   IF "Modbus_Buffer".Time_Venting <> 0 AND "Modbus_Buffer".Time_Venting <> "Torche_DB".Signal_Torche.Time_vent_g THEN
           "Torche_DB".Signal_Torche.Time_vent_g := "Modbus_Buffer".Time_Venting;
       END_IF;
       IF "Modbus_Buffer".Time_firing <> 0 AND "Modbus_Buffer".Time_firing <> "Torche_DB".Signal_Torche.Time_firing_g THEN
           "Torche_DB".Signal_Torche.Time_firing_g := "Modbus_Buffer".Time_firing;
       END_IF;
       IF "Modbus_Buffer".Time_spark_on <> 0 AND "Modbus_Buffer".Time_spark_on <> "Torche_DB".Signal_Torche.Time_spark_on_g THEN
           "Torche_DB".Signal_Torche.Time_spark_on_g := "Modbus_Buffer".Time_spark_on;
       END_IF;
       IF "Modbus_Buffer".Time_spark_off <> 0 AND "Modbus_Buffer".Time_spark_off <> "Torche_DB".Signal_Torche.Time_spark_off_g THEN
           "Torche_DB".Signal_Torche.Time_spark_off_g := "Modbus_Buffer".Time_spark_off;
       END_IF;
       IF "Modbus_Buffer".Time_stabil <> 0 AND "Modbus_Buffer".Time_stabil <> "Torche_DB".Signal_Torche.Time_stabiliz_g THEN
           "Torche_DB".Signal_Torche.Time_stabiliz_g := "Modbus_Buffer".Time_stabil;
       END_IF;
       IF "Modbus_Buffer".Time_after_alarm <> 0 AND "Modbus_Buffer".Time_after_alarm <> "Torche_DB".Signal_Torche.Time_after_alm_g  THEN
           "Torche_DB".Signal_Torche.Time_after_alm_g:= "Modbus_Buffer".Time_after_alarm;
       END_IF;
       IF "Modbus_Buffer".Time_after_stop <> 0 AND "Modbus_Buffer".Time_after_stop <> "Torche_DB".Signal_Torche.Time_stop_fire_g THEN
           "Torche_DB".Signal_Torche.Time_stop_fire_g := "Modbus_Buffer".Time_after_stop;
       END_IF;

       IF "Modbus_Buffer".Temp_Fire <> 0 AND "Modbus_Buffer".Temp_Fire <> "Temp_gorelka".Signal_AI.HH_Lim THEN
           "Temp_gorelka".Signal_AI.HH_Lim := "Modbus_Buffer".Temp_Fire;
       END_IF;
       IF "Modbus_Buffer".Temp_Fire <> 0 AND "Modbus_Buffer".Temp_Fire <> "temp_gorelka_2".Signal_AI.HH_Lim THEN
           "temp_gorelka_2".Signal_AI.HH_Lim := "Modbus_Buffer".Temp_Fire;
       END_IF;
       IF "Modbus_Buffer".Scal_max <> 0 AND "Modbus_Buffer".Scal_max <> "Temp_gorelka".Signal_AI.Scal_Max_Eu THEN
           "Temp_gorelka".Signal_AI.Scal_Max_Eu := "Modbus_Buffer".Scal_max;
       END_IF;
       IF "Modbus_Buffer".Scal_max <> 0 AND "Modbus_Buffer".Scal_max <> "temp_gorelka_2".Signal_AI.Scal_Max_Eu THEN
           "temp_gorelka_2".Signal_AI.Scal_Max_Eu := "Modbus_Buffer".Scal_max;
       END_IF;
       IF "Modbus_Buffer".Scal_min <> 0 AND "Modbus_Buffer".Scal_min <> "Temp_gorelka".Signal_AI.Scal_Min_Eu THEN
           "Temp_gorelka".Signal_AI.Scal_Min_Eu := "Modbus_Buffer".Scal_min;
       END_IF;
       IF "Modbus_Buffer".Scal_min <> 0 AND "Modbus_Buffer".Scal_min <> "temp_gorelka_2".Signal_AI.Scal_Min_Eu THEN
           "temp_gorelka_2".Signal_AI.Scal_Min_Eu := "Modbus_Buffer".Scal_min;
       END_IF;




   //********************ФОрмирование команды: запуск факела с верхнего уровня
   IF NOT "Modbus_Buffer".Start THEN
       "MB_Start" := false;
   ELSIF "Modbus_Buffer".Start THEN
       "MB_Start" := true;
       "Modbus_Buffer".Start := false;
   END_IF;

   IF NOT "Modbus_Buffer".Stop THEN
       "MB_Stop" := false;
   ELSIF "Modbus_Buffer".Stop THEN
       "MB_Stop" := true;
       "Modbus_Buffer".Stop := false;
   END_IF;

   IF NOT "Modbus_Buffer".Temp_curr_voltage THEN
       "Temp_gorelka".Signal_AI.VoltageInputType := false;
   ELSIF "Modbus_Buffer".Temp_curr_voltage THEN
       "Temp_gorelka".Signal_AI.VoltageInputType := true;
   END_IF;

   IF NOT "Modbus_Buffer".Temp_curr_voltage THEN
       "temp_gorelka_2".Signal_AI.VoltageInputType := false;
   ELSIF "Modbus_Buffer".Temp_curr_voltage THEN
       "temp_gorelka_2".Signal_AI.VoltageInputType := true;
   END_IF;
END_FUNCTION

// folder: PROFINET

FUNCTION "PUT" : Void   // FC9, SCL
{ S7_Optimized_Access := 'TRUE' }
VERSION : 0.1
BEGIN
   //"PN_XCHANGE_DB".AI1_Ch1 := "PT200".Signal_AI;
   //"PN_XCHANGE_DB".AI1_Ch2 := "TT200".Signal_AI;
   //"PN_XCHANGE_DB".AI1_Ch3 := "LT200_1".Signal_AI;
   //нужно дописать перемещение всех данных и заполнить PN_XCHANGE_DB
END_FUNCTION

FUNCTION "GET" : Void   // FC12, SCL
{ S7_Optimized_Access := 'TRUE' }
VERSION : 0.1
BEGIN
   //"PT200".Signal_AI := "PN_XCHANGE_DB".AI1_Ch1;
   // Заполнить до конца, разобраться когда вызывать эту функцию и функцию PUT
END_FUNCTION

FUNCTION "FC_SEND" : Void   // FC100, FBD
{ S7_Optimized_Access := 'TRUE' }
VERSION : 0.1
BEGIN

REGION Network 1
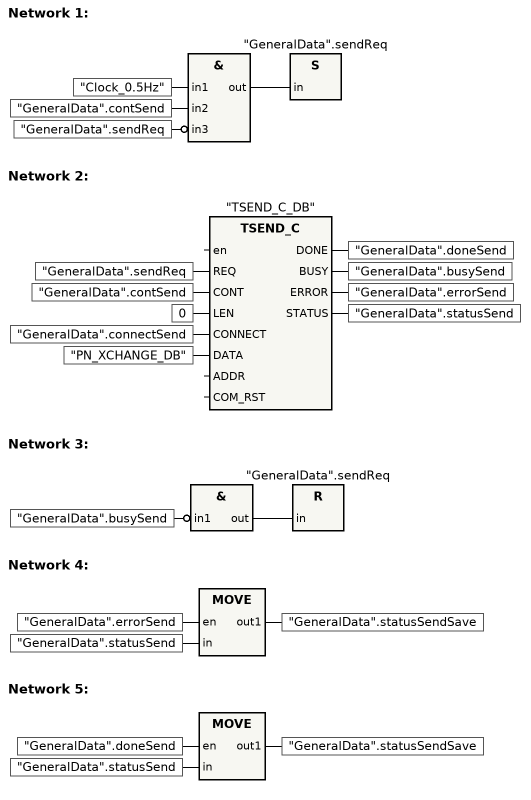
   IF "Clock_0.5Hz" AND "GeneralData".contSend AND NOT "GeneralData".sendReq THEN
       "GeneralData".sendReq := TRUE;
   END_IF;
END_REGION

REGION Network 2
   "TSEND_C_DB"(REQ := "GeneralData".sendReq,   // TSEND_C
                CONT := "GeneralData".contSend,
                LEN := 0,
                CONNECT := "GeneralData".connectSend,
                DATA := "PN_XCHANGE_DB",
                DONE => "GeneralData".doneSend,
                BUSY => "GeneralData".busySend,
                ERROR => "GeneralData".errorSend,
                STATUS => "GeneralData".statusSend);
END_REGION

REGION Network 3
   IF NOT "GeneralData".busySend THEN "GeneralData".sendReq := FALSE; END_IF;
END_REGION

REGION Network 4
   IF "GeneralData".errorSend THEN "GeneralData".statusSendSave := "GeneralData".statusSend; END_IF;
END_REGION

REGION Network 5
   IF "GeneralData".doneSend THEN "GeneralData".statusSendSave := "GeneralData".statusSend; END_IF;
END_REGION
END_FUNCTION

FUNCTION "FC_RECV" : Void   // FC200, FBD
{ S7_Optimized_Access := 'TRUE' }
VERSION : 0.1
BEGIN

REGION Network 1
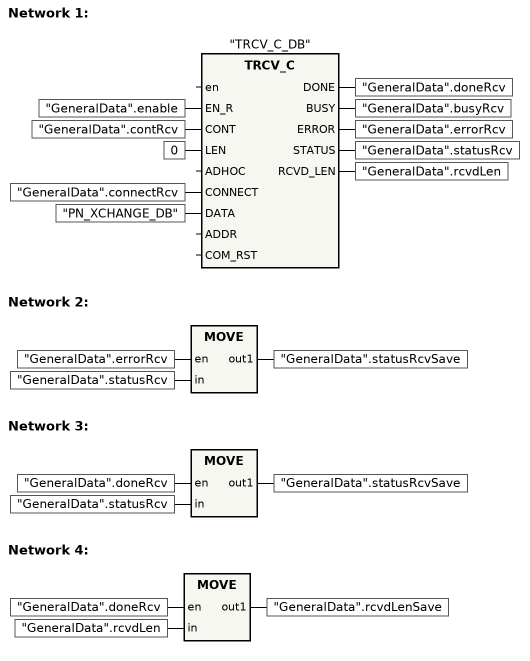
   "TRCV_C_DB"(EN_R := "GeneralData".enable,   // TRCV_C
               CONT := "GeneralData".contRcv,
               LEN := 0,
               CONNECT := "GeneralData".connectRcv,
               DATA := "PN_XCHANGE_DB",
               DONE => "GeneralData".doneRcv,
               BUSY => "GeneralData".busyRcv,
               ERROR => "GeneralData".errorRcv,
               STATUS => "GeneralData".statusRcv,
               RCVD_LEN => "GeneralData".rcvdLen);
END_REGION

REGION Network 2
   IF "GeneralData".errorRcv THEN "GeneralData".statusRcvSave := "GeneralData".statusRcv; END_IF;
END_REGION

REGION Network 3
   IF "GeneralData".doneRcv THEN "GeneralData".statusRcvSave := "GeneralData".statusRcv; END_IF;
END_REGION

REGION Network 4
   IF "GeneralData".doneRcv THEN "GeneralData".rcvdLenSave := "GeneralData".rcvdLen; END_IF;
END_REGION
END_FUNCTION